INTERFACE I_ProductionMode EXTENDS I_PackMLMode

END_INTERFACE

(* stored: Version 1.1.0.1, ProductVersion 3.1.4024.12
   Itf I_ProductionMode: Id {bdc8a500-a508-4eb5-927b-bbfe8257c22c} *)
